Staubli VAL3: SettingDET.dtx

num nCOLMAX = 39
num nCOLMIN
public num nColumn
public num nFocused
public num nListSize
num nROWMAX = 12
num nROWMIN
public num nRow
string sErrorMessage
string sErrorMsg[10]
  [1] = "An error has been detected in the Page library *\../*"
  [2] = "Variable sTxtBoxLen[*] has an illegal value"
  [3] = "Variable sTxtBoxPos[*] has an illegal value"
public string sFALSE = "FALSE"
public string sLabel = "-Detection ---"
public string sLabelPos = "0;0"
public string sMenu = "; GENERAL ; ENCODER ; CONVEYOR ; Ok"
public string sTRUE = "TRUE"
public string sTitle
public string sTxtBoxAuthord = "0123456789"
public string sTxtBoxCaption = "NbObject:"
public string sTxtBoxLen = "2"
public string sTxtBoxPos = "0;1"
public string sTxtBoxRange = "2;50"
public string sTxtBoxType = "N"
public string sTxtBoxVal = "1"
public string sListItem0
